(* CoDeSys 2.3.9.28 project: Aula08_ex1.pro *)
(* Libraries: Standard.lib 27.1.09 11:27:38, Util.lib 27.1.09 11:27:38, IecSfc.lib*24.11.08 08:07:15, SysLibTime.lib*27.1.09 11:27:38, SysTaskInfo.lib 24.11.08 08:07:15, SYSLIBCALLBACK.LIB 27.1.09 11:27:38 *)

(* PLC configuration (modules and I/O channels)
Hexswitch AT %IB0 [HexSwitch] rotary switch 0 = STOP, 1-15 = RUN
IOModules [CPX_MASTER] node 0, in %IB4 out %QB0
  8DI/8DO [CPX-8DI_8DO_Multi_I_O_module_1] node 0, in %IB4 out %QB0 {StringParam = 4,8,1,8,1; ByteParam = 7; ByteParam = 81; ByteParam = 0; ByteParam = 0; ByteParam = 0; ByteParam = 0; ByteParam = 0; IdleStateParam = 0; IdleModeParam = 255; IdleStateParam = 0; IdleModeParam = 255; IdleStateParam = 0; IdleModeParam = 255; IdleStateParam = 0; IdleModeParam = 255}
    AT %IB4 [ByteInput] -
    AT %QB0 [ByteOutput] -
  8DI/8DO [CPX-8DI_8DO_Multi_I_O_module_1] node 1, in %IB8 out %QB4 {StringParam = 4,8,1,8,1; ByteParam = 7; ByteParam = 81; ByteParam = 0; ByteParam = 0; ByteParam = 0; ByteParam = 0; ByteParam = 0; IdleStateParam = 0; IdleModeParam = 255; IdleStateParam = 0; IdleModeParam = 255; IdleStateParam = 0; IdleModeParam = 255; IdleStateParam = 0; IdleModeParam = 255}
    AT %IB8 [ByteInput] -
    AT %QB4 [ByteOutput] -
*)

(* Global variable list: Global_Variables *)
VAR_GLOBAL

	START AT %IX2.0 : BOOL;
	STOP AT %IX2.1 : BOOL;
	S1 AT %IX2.2 : BOOL;
	S2 AT %IX2.3 : BOOL;
	S3 AT %IX2.4 : BOOL;

	M1 AT %QX0.0 : BOOL;
	LP AT %QX0.1 : BOOL;
	C1 AT %QX0.2 : BOOL;
	V1 AT %QX0.3 : BOOL;

	MEM : BOOL;
	MEM2: BOOL;
	MEM3 : BOOL;

	T1 : TON;
	T2 : TON;
	T3 : TON;

END_VAR

(* POU PLC_PRG, LD *)
PROGRAM PLC_PRG
VAR
END_VAR
VAR (* helpers for the ST form of the networks *)
	_p1 : BOOL;
END_VAR
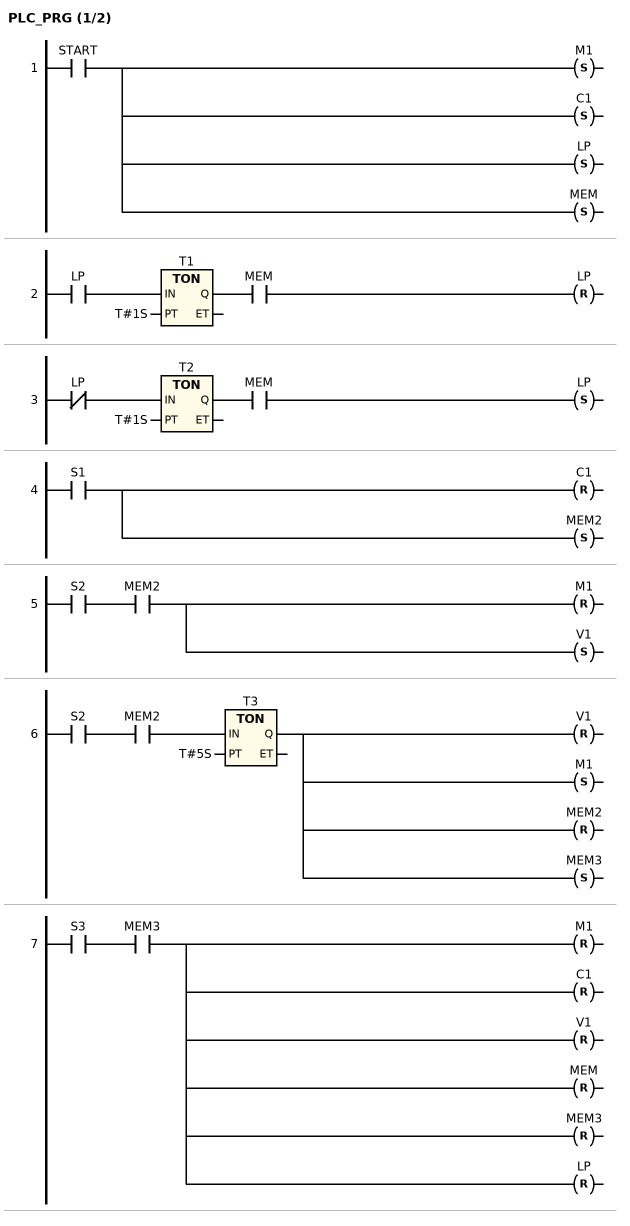
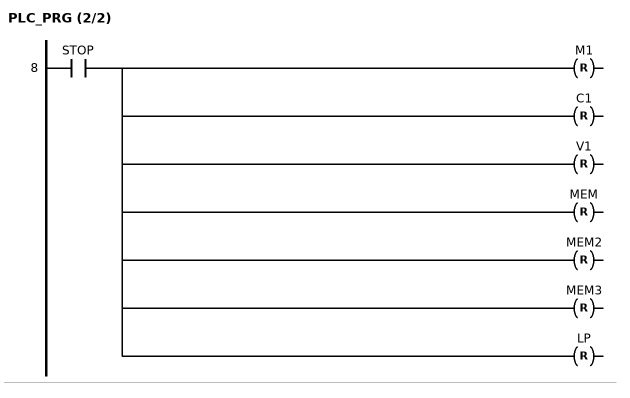
_LD_ (* Ladder Diagram *)
NETWORK 1
	[START] --- (S M1) (S C1) (S LP) (S MEM)
NETWORK 2
	[LP] - T1:TON(IN: *, PT: T#1S) - [MEM] --- (R LP)
NETWORK 3
	[/LP] - T2:TON(IN: *, PT: T#1S) - [MEM] --- (S LP)
NETWORK 4
	[S1] --- (R C1) (S MEM2)
NETWORK 5
	[S2] - [MEM2] --- (R M1) (S V1)
NETWORK 6
	[S2] - [MEM2] - T3:TON(IN: *, PT: T#5S) --- (R V1) (S M1) (R MEM2) (S MEM3)
NETWORK 7
	[S3] - [MEM3] --- (R M1) (R C1) (R V1) (R MEM) (R MEM3) (R LP)
NETWORK 8
	[STOP] --- (R M1) (R C1) (R V1) (R MEM) (R MEM2) (R MEM3) (R LP)
_END_LD_
(* the same logic as Structured Text *)
(* Network 1 *)
IF START THEN M1 := TRUE; C1 := TRUE; LP := TRUE; MEM := TRUE; END_IF;
(* Network 2 *)
T1(IN := LP, PT := T#1S);
IF T1.Q AND MEM THEN LP := FALSE; END_IF;
(* Network 3 *)
T2(IN := NOT LP, PT := T#1S);
IF T2.Q AND MEM THEN LP := TRUE; END_IF;
(* Network 4 *)
IF S1 THEN C1 := FALSE; MEM2 := TRUE; END_IF;
(* Network 5 *)
IF S2 AND MEM2 THEN M1 := FALSE; V1 := TRUE; END_IF;
(* Network 6 *)
T3(IN := S2 AND MEM2, PT := T#5S);
IF T3.Q THEN V1 := FALSE; M1 := TRUE; MEM2 := FALSE; MEM3 := TRUE; END_IF;
(* Network 7 *)
_p1 := S3 AND MEM3;
IF _p1 THEN M1 := FALSE; C1 := FALSE; V1 := FALSE; MEM := FALSE; MEM3 := FALSE; LP := FALSE; END_IF;
(* Network 8 *)
IF STOP THEN M1 := FALSE; C1 := FALSE; V1 := FALSE; MEM := FALSE; MEM2 := FALSE; MEM3 := FALSE; LP := FALSE; END_IF;
END_PROGRAM
